{attribute 'GeneratedUsingTerminal: KL1512'}
{attribute addProperty BoxType "KL1512"}
{attribute addProperty Id "StateAT %I*USINT0Data_InAT %I*UINT0CtrlAT %Q*USINT0Data_OutAT %Q*UINT0"}
{attribute addProperty CRC "63875678"}
{attribute addProperty Size "0"}
TYPE Channel_03CEAA5E :
STRUCT
	{attribute addProperty Name "State"}
	State AT %I* : USINT;
	{attribute addProperty Name "Data_In"}
	Data_In AT %I* : UINT;
	{attribute addProperty Name "Ctrl"}
	Ctrl AT %Q* : USINT;
	{attribute addProperty Name "Data_Out"}
	Data_Out AT %Q* : UINT;
END_STRUCT
END_TYPE

(* stored: Version 1.2.0.0, ProductVersion 3.1.4024.11
   DUT Channel_03CEAA5E: Id {b32732e8-1161-4bba-ab7d-7f3d7ecfa999} *)
